FUNCTION_BLOCK PUBLIC GearInCA  IMPLEMENTS I_Task
VAR
	GearInPosCA : Tc3_McCollisionAvoidance.MC_GearInPosCA;
	_syncStrategy : Tc3_Mc3Definitions.MC_SYNC_STRATEGY := Tc3_Mc3Definitions.MC_SYNC_STRATEGY.mcSyncStrategyEarly;
	_SlaveAxis : REFERENCE TO Tc2_MC2.AXIS_REF;
	_MasterAxis : REFERENCE TO Tc2_MC2.AXIS_REF;
	_GearMover: BOOL;
	_ErrorID: UDINT;
		State: INT;
	_Done: BOOL;
	_Error: BOOL;
	_Busy: BOOL;
END_VAR

{analysis -2}

METHOD Abort : BOOL
GearInPosCA.Execute := FALSE;
_GearMover := FALSE;
_Busy := false;
Abort := true;
State := 0;
END_METHOD

PROPERTY Busy : BOOL
GET
Busy := _Busy;
END_GET
END_PROPERTY

METHOD Cycle : HRESULT
VAR_INPUT
END_VAR
Cycle := S_OK;
CASE State OF
	0:
		IF _GearMover THEN
			Cycle := S_PENDING;
			_Done := FALSE;
			_Error := FALSE;
			_Busy := TRUE;
			GearInPosCA.Execute := TRUE;
			IF GearInPosCA.Busy THEN
				State := 10;
				_GearMover := FALSE;
			END_IF
		END_IF
		
	10:
		IF GearInPosCA.InSync THEN
			GearInPosCA.Execute := FALSE;
			_Busy := FALSE;
			_Done := TRUE;
			State := 0;
			Cycle := S_OK;
		END_IF
	ELSE
		Cycle := E_FAIL;
END_CASE
_Error := GearInPosCA.Error;
_ErrorID := GearInPosCA.ErrorId;
IF __ISVALIDREF(_MasterAxis) AND __ISVALIDREF(_SlaveAxis) THEN
	GearInPosCA(Master := _MasterAxis, Slave := _SlaveAxis, SyncStrategy := _syncStrategy, Velocity := 2000.0, RatioNumerator := 1, Gap := 60.0);
END_IF
END_METHOD

PROPERTY Done : BOOL
GET
Done := _Done;
END_GET
END_PROPERTY

PROPERTY Error : BOOL
GET
Error := _Error;
END_GET
END_PROPERTY

METHOD FB_init : BOOL
VAR_INPUT
	bInitRetains : BOOL; // if TRUE, the retain variables are initialized (warm start / cold start)
	bInCopyCode : BOOL;  // if TRUE, the instance afterwards gets moved into the copy code (online change)
	axis : reference TO AXIS_REF;
END_VAR
_SlaveAxis REF= axis;
END_METHOD

PROPERTY MyGearMaster : REFERENCE TO AXIS_REF
GET
MyGearMaster REF= _MasterAxis;
END_GET
SET
_MasterAxis REF= MyGearMaster;
END_SET
END_PROPERTY

METHOD PUBLIC Sync : BOOL
VAR_INPUT
	MasterPosition : MC_LREAL;
	SlavePosition : MC_LREAL;
END_VAR
GearInPosCA.MasterSyncPosition := MasterPosition;
GearInPosCA.SlaveSyncPosition := SlavePosition;
_GearMover := Sync := true;
END_METHOD

PROPERTY PUBLIC SyncStrategy : mc_sync_strategy
GET
SyncStrategy := _syncStrategy;
END_GET
SET
_syncStrategy := SyncStrategy;
END_SET
END_PROPERTY

END_FUNCTION_BLOCK

(* stored: Version 1.1.0.1
   POU GearInCA: Id {4eabfc6f-0e0b-4cf2-8798-42f7d613e2e0}, SpecialFunc None
   Method Abort: Id {33a44f0c-0e3b-4808-ac44-6bb8acc99a21}
   Property Busy: Id {4b87a8a5-0488-49e9-9c97-79ee531d0f30}
   Get Get: Id {ae7f8c84-bd44-4377-ac93-c5e80d9322fd}
   Method Cycle: Id {63d39597-d1df-4364-9e4b-a587d0a782e8}
   Property Done: Id {4ec2e7b3-ecd4-4788-b9d1-484eeb59988f}
   Get Get: Id {870c3b62-4cf2-4c56-9b9c-d05cf4fbc241}
   Property Error: Id {b0cd652d-d067-40fd-9e01-a5029b2c46d5}
   Get Get: Id {3fb8f055-5da1-4e27-bc19-18113abf4bbd}
   Method FB_init: Id {3fc0c81f-a0ab-4736-b340-c6d7f16fcfa0}
   Property MyGearMaster: Id {a46ef8fb-4e90-4897-9dcd-a04c2dd2e88d}
   Get Get: Id {e800e4fe-3c89-421e-9396-ebf9ce3426e8}
   Set Set: Id {8696c54d-0b3c-4ca7-832b-6895b239a418}
   Method Sync: Id {3bab61dc-be16-4255-9286-dba4fcc8047d}
   Property SyncStrategy: Id {74227846-5fda-4bbe-ac22-10f463d682ca}
   Get Get: Id {1146c154-913b-407f-8846-59691fdc56f4}
   Set Set: Id {42d81a91-d986-4985-a960-1c593b4fd69b} *)
